(* IEC 61131-3 sources: Industry-PLC-LLM/data/PLCBEAD_repo/PLCBEAD_PLCEmbed-main/PLC-BEAD/Source/GEB/COSH, 1 file *)

(* ---- COSH.ST ---- *)
FUNCTION COSH:REAL
	VAR_INPUT
		X :	REAL;
	END_VAR

	VAR
		T :	REAL;
	END_VAR

	T := EXP(X);
	COSH := (1.0 / T + T) * 0.5;
END_FUNCTION

PROGRAM program0
  VAR
    LocalVar0 : REAL;
    CEIL5_OUT : REAL;
  END_VAR

  CEIL5_OUT := COSH(LocalVar0);
END_PROGRAM
